{attribute addProperty BoxType "EL5001-0090-0016"}
{attribute addProperty Id "Data_errorBIT10.1251Frame_errorBIT10.1252Power_failureBIT10.1253Sync_errorBIT10.12514TxPDO_StateBIT10.12515TxPDO_ToggleBIT10.12516"}
{attribute addProperty CRC "4018601410"}
{attribute addProperty SizeInBites "16"}
{attribute addProperty SizeInBytes "2"}
TYPE Status_EF86FDC2 :
STRUCT
	{attribute addProperty Name "Data_error"}
	Data_error : BIT;
	{attribute addProperty Name "Frame_error"}
	Frame_error : BIT;
	{attribute addProperty Name "Power_failure"}
	Power_failure : BIT;
	{attribute 'hide'}
	reserve_1_BIT_0 : BIT;
	{attribute 'hide'}
	reserve_1_BIT_1 : BIT;
	{attribute 'hide'}
	reserve_1_BIT_2 : BIT;
	{attribute 'hide'}
	reserve_1_BIT_3 : BIT;
	{attribute 'hide'}
	reserve_1_BIT_4 : BIT;
	{attribute 'hide'}
	reserve_1_BIT_5 : BIT;
	{attribute 'hide'}
	reserve_1_BIT_6 : BIT;
	{attribute 'hide'}
	reserve_1_BIT_7 : BIT;
	{attribute 'hide'}
	reserve_1_BIT_8 : BIT;
	{attribute 'hide'}
	reserve_1_BIT_9 : BIT;
	{attribute addProperty Name "Sync_error"}
	Sync_error : BIT;
	{attribute addProperty Name "TxPDO_State"}
	TxPDO_State : BIT;
	{attribute addProperty Name "TxPDO_Toggle"}
	TxPDO_Toggle : BIT;
END_STRUCT
END_TYPE

(* stored: Version 1.2.0.0, ProductVersion 3.1.4024.9
   DUT Status_EF86FDC2: Id {a07c0cf8-3901-430e-9292-79567b64abc3} *)
